PROGRAM MAIN
VAR
END_VAR

END_PROGRAM

(* stored: Version 1.1.0.1, ProductVersion 3.1.4024.11
   POU MAIN: Id {865bfc75-0015-4a63-8a3f-abd23effa663}, SpecialFunc None *)
